FUNCTION_BLOCK PUBLIC QueueForwardEnumerator_TestSuite EXTENDS TcUnit.FB_TestSuite

CheckIsValidAtStart();
CheckMoveNextReturnsFalseAtTheEnd();
CheckMoveNextReturnsFalseWhenEmpty();
CheckMoveNextReturnsTrueMultipleItems();
CheckMoveNextReturnsTrueSingleItem();
CheckReset();
CheckTryGet();
CheckTryGetTo();
CheckWorksWithIntegers();
CheckWorksWithStrings();
CheckWorksWithArrays();

METHOD PUBLIC CheckIsValidAtStart
VAR
	result : BOOL;
	queue : Queue;
	enumerator : I_ForwardEnumerator;
END_VAR
TEST('CheckIsValidAtStart');

enumerator := queue.GetEnumerator();

result := enumerator.IsValid;
enumerator.Dispose();

AssertTrue(
	Condition := result,
	Message := 'Method returned false'
);

TEST_FINISHED();
END_METHOD

METHOD PRIVATE CheckMoveNextReturnsFalseAtTheEnd
VAR
	in1 : INT := 123;
	result : BOOL;
	queue : Queue;
	enumerator : I_ForwardEnumerator;
END_VAR
TEST('CheckMoveNextReturnsFalseAtTheEnd');

queue.Enqueue(in1);
enumerator := queue.GetEnumerator();

enumerator.MoveNext();
result := enumerator.MoveNext();
enumerator.Dispose();

AssertFalse(result,
    'MoveNext did not correctly signal the end of the enumeration');
	
TEST_FINISHED();
END_METHOD

METHOD PUBLIC CheckMoveNextReturnsFalseWhenEmpty
VAR
	result : BOOL;
	queue : Queue;
	enumerator : I_ForwardEnumerator;
END_VAR
TEST('CheckMoveNextReturnsFalseWhenEmpty');

enumerator := queue.GetEnumerator();

result := enumerator.MoveNext();
enumerator.Dispose();

AssertFalse(
	Condition := result,
	Message := 'MoveNext did not correctly signal the end of the enumeration'
);

TEST_FINISHED();
END_METHOD

METHOD PRIVATE CheckMoveNextReturnsTrueMultipleItems
VAR
	in1 : INT := 123;
	in2 : INT := 456;
	in3 : INT := 789;
	result : BOOL;
	queue : Queue;
	enumerator : I_ForwardEnumerator;
END_VAR
TEST('CheckMoveNextReturnsTrueMultipleItems');

queue.Enqueue(in1);
queue.Enqueue(in2);
queue.Enqueue(in3);
enumerator := queue.GetEnumerator();

result := enumerator.MoveNext();
enumerator.Dispose();

AssertTrue(result, 'MoveNext did not correctly signal there were more items to follow');

TEST_FINISHED();
END_METHOD

METHOD PRIVATE CheckMoveNextReturnsTrueSingleItem
VAR
	in1 : INT := 123;
	result : BOOL;
	queue : Queue;
	enumerator : I_ForwardEnumerator;
END_VAR
TEST('CheckMoveNextReturnsTrueSingleItem');

queue.Enqueue(in1);
enumerator := queue.GetEnumerator();

result := enumerator.MoveNext();
enumerator.Dispose();

AssertTrue(result,
    'MoveNext did not correctly signal there were more items to follow');
	
TEST_FINISHED();
END_METHOD

METHOD PUBLIC CheckReset
VAR
	in1 : ARRAY [0..1] OF REAL := [0.1,2.3];
	in2 : ARRAY [0..1] OF REAL := [1.2,3.4];
	in3 : ARRAY [0..1] OF REAL := [2.3,4.5];
	out : ARRAY [0..1] OF REAL;
	expected : ARRAY [0..1] OF REAL := [0.1,2.3];
	queue : Queue;
	enumerator : I_ForwardEnumerator;
END_VAR
TEST('CheckReset');

queue.Enqueue(in1);
queue.Enqueue(in2);
queue.Enqueue(in3);

enumerator := queue.GetEnumerator();

enumerator.MoveNext();
enumerator.MoveNext();
enumerator.Reset();
enumerator.MoveNext();
enumerator.TryGet(out);

enumerator.Dispose();

AssertEquals(
	Expected := expected,
	Actual := out,
	Message := 'Did not produce the expected result'
);

TEST_FINISHED();
END_METHOD

METHOD PUBLIC CheckTryGet
VAR
	in : INT := 123;
	out : INT;
	expected : INT := 123;
	result : BOOL;
	queue : Queue;
	enumerator : I_ForwardEnumerator;
END_VAR
TEST('CheckTryGet');

queue.Enqueue(in);
enumerator := queue.GetEnumerator();
enumerator.MoveNext();

result := enumerator.TryGet(out);
enumerator.Dispose();

AssertTrue(
	Condition := result,
	Message := 'Method returned false'
);

AssertEquals(
	Expected := expected,
	Actual := out,
	Message := 'Did not produce the expected result'
);

TEST_FINISHED();
END_METHOD

METHOD PUBLIC CheckTryGetTo
VAR
	in : INT := 123;
	out : INT;
	expected : INT := 123;
	result : BOOL;
	queue : Queue;
	enumerator : I_ForwardEnumerator;
END_VAR
TEST('CheckTryGetTo');

queue.Enqueue(in);
enumerator := queue.GetEnumerator();
enumerator.MoveNext();

result := enumerator.TryGetTo(ADR(out),SIZEOF(out));
enumerator.Dispose();

AssertTrue(
	Condition := result,
	Message := 'Method returned false'
);

AssertEquals(
	Expected := expected,
	Actual := out,
	Message := 'Did not produce the expected result'
);

TEST_FINISHED();
END_METHOD

METHOD PUBLIC CheckWorksWithArrays
VAR
	in1 : ARRAY [0..1] OF REAL := [0.1,2.3];
	in2 : ARRAY [0..1] OF REAL := [1.2,3.4];
	in3 : ARRAY [0..1] OF REAL := [2.3,4.5];
	out1 : ARRAY [0..1] OF REAL;
	out2 : ARRAY [0..1] OF REAL;
	out3 : ARRAY [0..1] OF REAL;
	expected1 : ARRAY [0..1] OF REAL := [0.1,2.3];
	expected2 : ARRAY [0..1] OF REAL := [1.2,3.4];
	expected3 : ARRAY [0..1] OF REAL := [2.3,4.5];
	queue : Queue;
	enumerator : I_ForwardEnumerator;
END_VAR
TEST('CheckWorksWithArrays');

queue.Enqueue(in1);
queue.Enqueue(in2);
queue.Enqueue(in3);

enumerator := queue.GetEnumerator();

enumerator.MoveNext();
enumerator.TryGet(out1);
enumerator.MoveNext();
enumerator.TryGet(out2);
enumerator.MoveNext();
enumerator.TryGet(out3);

enumerator.Dispose();

AssertEquals(
	Expected := expected1,
	Actual := out1,
	Message := 'Did not produce the expected 1st result'
);

AssertEquals(
	Expected := expected2,
	Actual := out2,
	Message := 'Did not produce the expected 2nd result'
);

AssertEquals(
	Expected := expected3,
	Actual := out3,
	Message := 'Did not produce the expected 3rd result'
);

TEST_FINISHED();
END_METHOD

METHOD PUBLIC CheckWorksWithIntegers
VAR
	in1 : INT := 123;
	in2 : INT := 234;
	in3 : INT := 345;
	out1 : INT;
	out2 : INT;
	out3 : INT;
	expected1 : INT := 123;
	expected2 : INT := 234;
	expected3 : INT := 345;
	queue : Queue;
	enumerator : I_ForwardEnumerator;
END_VAR
TEST('CheckWorksWithIntegers');

queue.Enqueue(in1);
queue.Enqueue(in2);
queue.Enqueue(in3);

enumerator := queue.GetEnumerator();

enumerator.MoveNext();
enumerator.TryGet(out1);
enumerator.MoveNext();
enumerator.TryGet(out2);
enumerator.MoveNext();
enumerator.TryGet(out3);

enumerator.Dispose();

AssertEquals(
	Expected := expected1,
	Actual := out1,
	Message := 'Did not produce the expected 1st result'
);

AssertEquals(
	Expected := expected2,
	Actual := out2,
	Message := 'Did not produce the expected 2nd result'
);

AssertEquals(
	Expected := expected3,
	Actual := out3,
	Message := 'Did not produce the expected 3rd result'
);

TEST_FINISHED();
END_METHOD

METHOD PUBLIC CheckWorksWithStrings
VAR
	in1 : STRING := 'test1';
	in2 : STRING := 'test2';
	in3 : STRING := 'test3';
	out1 : STRING;
	out2 : STRING;
	out3 : STRING;
	expected1 : STRING := 'test1';
	expected2 : STRING := 'test2';
	expected3 : STRING := 'test3';
	queue : Queue;
	enumerator : I_ForwardEnumerator;
END_VAR
TEST('CheckWorksWithStrings');

queue.Enqueue(in1);
queue.Enqueue(in2);
queue.Enqueue(in3);

enumerator := queue.GetEnumerator();

enumerator.MoveNext();
enumerator.TryGet(out1);
enumerator.MoveNext();
enumerator.TryGet(out2);
enumerator.MoveNext();
enumerator.TryGet(out3);

enumerator.Dispose();

AssertEquals(
	Expected := expected1,
	Actual := out1,
	Message := 'Did not produce the expected 1st result'
);

AssertEquals(
	Expected := expected2,
	Actual := out2,
	Message := 'Did not produce the expected 2nd result'
);

AssertEquals(
	Expected := expected3,
	Actual := out3,
	Message := 'Did not produce the expected 3rd result'
);

TEST_FINISHED();
END_METHOD

END_FUNCTION_BLOCK

(* stored: Version 1.1.0.1, ProductVersion 3.1.4024.12
   POU QueueForwardEnumerator_TestSuite: Id {9d1a4f2e-078d-0792-3403-40123a2b69ae}, SpecialFunc None
   Method CheckIsValidAtStart: Id {16a11caa-93f7-05d7-163a-35a9f3279dee}
   Method CheckMoveNextReturnsFalseAtTheEnd: Id {6f8f4f02-cbf1-0f34-16dd-867595333bbc}
   Method CheckMoveNextReturnsFalseWhenEmpty: Id {d8d2c804-0293-0076-37b3-0561a22ee557}
   Method CheckMoveNextReturnsTrueMultipleItems: Id {21ec4dd9-e4ce-0749-3aaf-287b0acf429f}
   Method CheckMoveNextReturnsTrueSingleItem: Id {f5266c4b-4efe-0898-1bdc-b57b0528db40}
   Method CheckReset: Id {1d0af406-04fe-0a63-0cef-0195bb712221}
   Method CheckTryGet: Id {90acc4fd-cd01-0949-0b91-bedce2361ffc}
   Method CheckTryGetTo: Id {d3a8529f-7ed6-0ed3-22c8-fb7827677c23}
   Method CheckWorksWithArrays: Id {51bdc2a7-25b2-040c-35b0-cbb38a1d3b21}
   Method CheckWorksWithIntegers: Id {75f82f32-3749-0496-0b65-4b20c0af7f7b}
   Method CheckWorksWithStrings: Id {1417836e-e0dc-0217-377b-65f8faa438e9} *)
